Universal Robots PolyScope program: welding.urp

Program welding (installation=default directory=/home/ur/ursim-current/programs createdIn=5.14.0 lastSavedIn=5.14.0 robotSerialNumber=20195299999)
Calibrated DH parameters: a=[0, -0.6127, -0.57155, 0, 0, 0]; d=[0.1807, 0, 0, 0.17415, 0.11985, 0.11655]; alpha=[1.570796, 0, 0, 1.570796, -1.570796, 0]; deltaTheta=[0, 0, 0, 0, 0, 0]
InitVariablesNode
BeforeStart
  test := True
  status := "READY"
  velocity := 10
Robot Program (runOnlyOnce=false)
  URCap HMI (Robpod HMI URcap, Robpod Cloud) dataModel(robpod.hmi.stop.main.loop=true, robpod.hmi.selected=/home/ur/ursim-current/programs/welding.hmi)
SubProgram weld_linear (keepSynchronizedWithDisk=false)
  status := "APPROACH"
  MoveJ speed 60 deg/s, acceleration 80 deg/s^2 (useActiveTCP=true positionType=JointAngles) feature=Base
    Waypoint Variable (Variable): variable=ApproachPose
  MoveL speed 250 mm/s, acceleration 1200 mm/s^2 (useActiveTCP=true) feature=Base
    Waypoint Variable (Variable): variable=ArcStartPose
  status := "WELDING"
  If not test
    Set DigitalOutput pin=digital_out[1]; digitalValue=1
  Script: movel(ArcEndPose, v=velocity/1000)
  Set DigitalOutput pin=digital_out[1]; digitalValue=0
  status := "RETRACT"
  MoveL speed 250 mm/s, acceleration 1200 mm/s^2 (useActiveTCP=true) feature=Base
    Waypoint Variable (Variable): variable=RetractPose
  status := "READY"
SubProgram weld_circular (keepSynchronizedWithDisk=false)
  status := "APPROACH"
  MoveJ speed 60 deg/s, acceleration 80 deg/s^2 (useActiveTCP=true positionType=JointAngles) feature=Base
    Waypoint Variable (Variable): variable=ApproachPose
  MoveL speed 250 mm/s, acceleration 1200 mm/s^2 (useActiveTCP=true) feature=Base
    Waypoint Variable (Variable): variable=ArcStartPose
  status := "WELDING"
  If not test
    Set DigitalOutput pin=digital_out[1]; digitalValue=1
  Script: movec(WaypointPose, ArcEndPose, v=velocity/1000)
  Set DigitalOutput pin=digital_out[1]; digitalValue=0
  status := "RETRACT"
  MoveL speed 250 mm/s, acceleration 1200 mm/s^2 (useActiveTCP=true) feature=Base
    Waypoint Variable (Variable): variable=RetractPose
  status := "READY"
